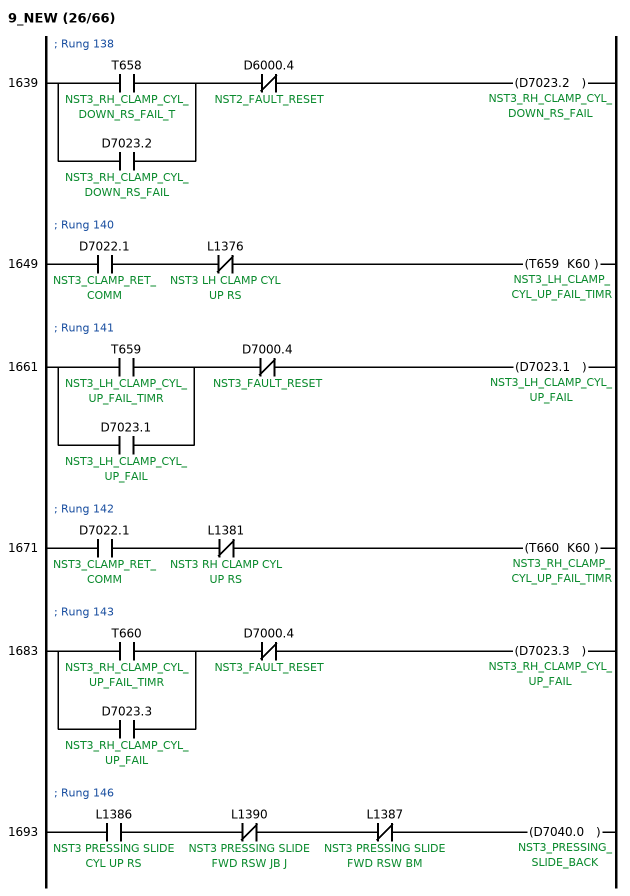
[picture p144: ladder of 9_NEW, rungs at steps 1639 to 1693]
; Rung 138
1639  LD      T658  ; NST3_RH_CLAMP_CYL_DOWN_RS_FAIL_T
      OR      D7023.2  ; NST3_RH_CLAMP_CYL_DOWN_RS_FAIL
      ANI     D6000.4  ; NST2_FAULT_RESET
      OUT     D7023.2  ; NST3_RH_CLAMP_CYL_DOWN_RS_FAIL
; Rung 140
1649  LD      D7022.1  ; NST3_CLAMP_RET_COMM
      ANI     L1376  ; NST3 LH CLAMP CYL UP RS
      OUT     T659 K60  ; NST3_LH_CLAMP_CYL_UP_FAIL_TIMR
; Rung 141
1661  LD      T659  ; NST3_LH_CLAMP_CYL_UP_FAIL_TIMR
      OR      D7023.1  ; NST3_LH_CLAMP_CYL_UP_FAIL
      ANI     D7000.4  ; NST3_FAULT_RESET
      OUT     D7023.1  ; NST3_LH_CLAMP_CYL_UP_FAIL
; Rung 142
1671  LD      D7022.1  ; NST3_CLAMP_RET_COMM
      ANI     L1381  ; NST3 RH CLAMP CYL UP RS
      OUT     T660 K60  ; NST3_RH_CLAMP_CYL_UP_FAIL_TIMR
; Rung 143
1683  LD      T660  ; NST3_RH_CLAMP_CYL_UP_FAIL_TIMR
      OR      D7023.3  ; NST3_RH_CLAMP_CYL_UP_FAIL
      ANI     D7000.4  ; NST3_FAULT_RESET
      OUT     D7023.3  ; NST3_RH_CLAMP_CYL_UP_FAIL
; Rung 146
1693  LD      L1386  ; NST3 PRESSING SLIDE CYL UP RS
      ANI     L1390  ; NST3 PRESSING SLIDE FWD RSW JB J
      ANI     L1387  ; NST3 PRESSING SLIDE FWD RSW BM
      OUT     D7040.0  ; NST3_PRESSING_SLIDE_BACK
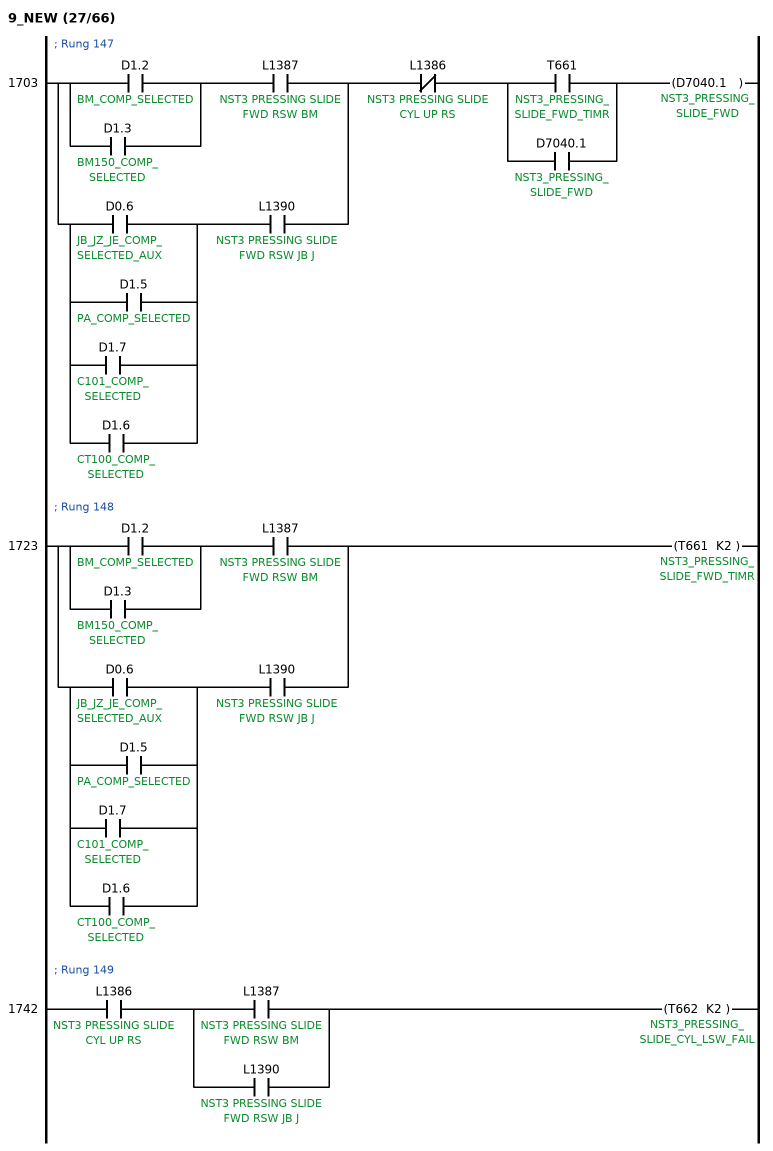
; Rung 147
1703  LD      D1.2  ; BM_COMP_SELECTED
      OR      D1.3  ; BM150_COMP_SELECTED
      AND     L1387  ; NST3 PRESSING SLIDE FWD RSW BM
      LD      D0.6  ; JB_JZ_JE_COMP_SELECTED_AUX
      OR      D1.5  ; PA_COMP_SELECTED
      OR      D1.7  ; C101_COMP_SELECTED
      OR      D1.6  ; CT100_COMP_SELECTED
      AND     L1390  ; NST3 PRESSING SLIDE FWD RSW JB J
      ORB
      ANI     L1386  ; NST3 PRESSING SLIDE CYL UP RS
      LD      T661  ; NST3_PRESSING_SLIDE_FWD_TIMR
      OR      D7040.1  ; NST3_PRESSING_SLIDE_FWD
      ANB
      OUT     D7040.1  ; NST3_PRESSING_SLIDE_FWD
; Rung 148
1723  LD      D1.2  ; BM_COMP_SELECTED
      OR      D1.3  ; BM150_COMP_SELECTED
      AND     L1387  ; NST3 PRESSING SLIDE FWD RSW BM
      LD      D0.6  ; JB_JZ_JE_COMP_SELECTED_AUX
      OR      D1.5  ; PA_COMP_SELECTED
      OR      D1.7  ; C101_COMP_SELECTED
      OR      D1.6  ; CT100_COMP_SELECTED
      AND     L1390  ; NST3 PRESSING SLIDE FWD RSW JB J
      ORB
      OUT     T661 K2  ; NST3_PRESSING_SLIDE_FWD_TIMR
; Rung 149
1742  LD      L1386  ; NST3 PRESSING SLIDE CYL UP RS
      LD      L1387  ; NST3 PRESSING SLIDE FWD RSW BM
      OR      L1390  ; NST3 PRESSING SLIDE FWD RSW JB J
      ANB
      OUT     T662 K2  ; NST3_PRESSING_SLIDE_CYL_LSW_FAIL
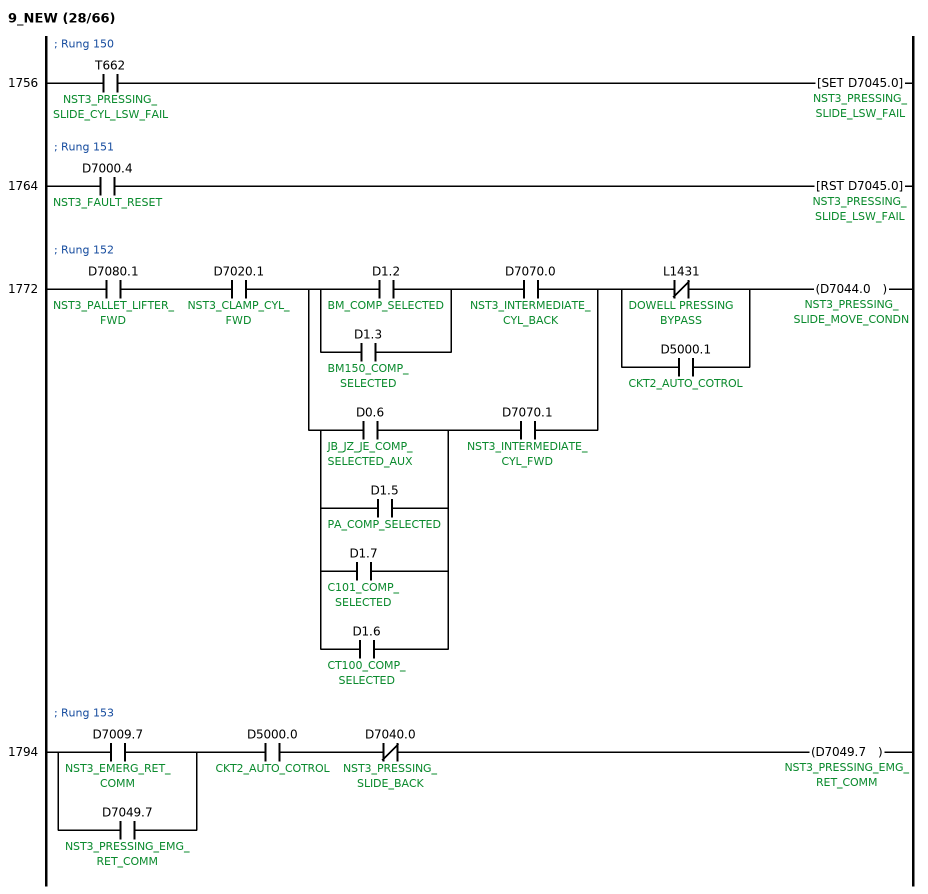
; Rung 150
1756  LD      T662  ; NST3_PRESSING_SLIDE_CYL_LSW_FAIL
      SET     D7045.0  ; NST3_PRESSING_SLIDE_LSW_FAIL
; Rung 151
1764  LD      D7000.4  ; NST3_FAULT_RESET
      RST     D7045.0  ; NST3_PRESSING_SLIDE_LSW_FAIL
; Rung 152
1772  LD      D7080.1  ; NST3_PALLET_LIFTER_FWD
      AND     D7020.1  ; NST3_CLAMP_CYL_FWD
      LD      D1.2  ; BM_COMP_SELECTED
      OR      D1.3  ; BM150_COMP_SELECTED
      AND     D7070.0  ; NST3_INTERMEDIATE_CYL_BACK
      LD      D0.6  ; JB_JZ_JE_COMP_SELECTED_AUX
      OR      D1.5  ; PA_COMP_SELECTED
      OR      D1.7  ; C101_COMP_SELECTED
      OR      D1.6  ; CT100_COMP_SELECTED
      AND     D7070.1  ; NST3_INTERMEDIATE_CYL_FWD
      ORB
      ANB
      LDI     L1431  ; DOWELL PRESSING BYPASS
      OR      D5000.1  ; CKT2_AUTO_COTROL
      ANB
      OUT     D7044.0  ; NST3_PRESSING_SLIDE_MOVE_CONDN
; Rung 153
1794  LD      D7009.7  ; NST3_EMERG_RET_COMM
      OR      D7049.7  ; NST3_PRESSING_EMG_RET_COMM
      AND     D5000.0  ; CKT2_AUTO_COTROL
      ANI     D7040.0  ; NST3_PRESSING_SLIDE_BACK
      OUT     D7049.7  ; NST3_PRESSING_EMG_RET_COMM
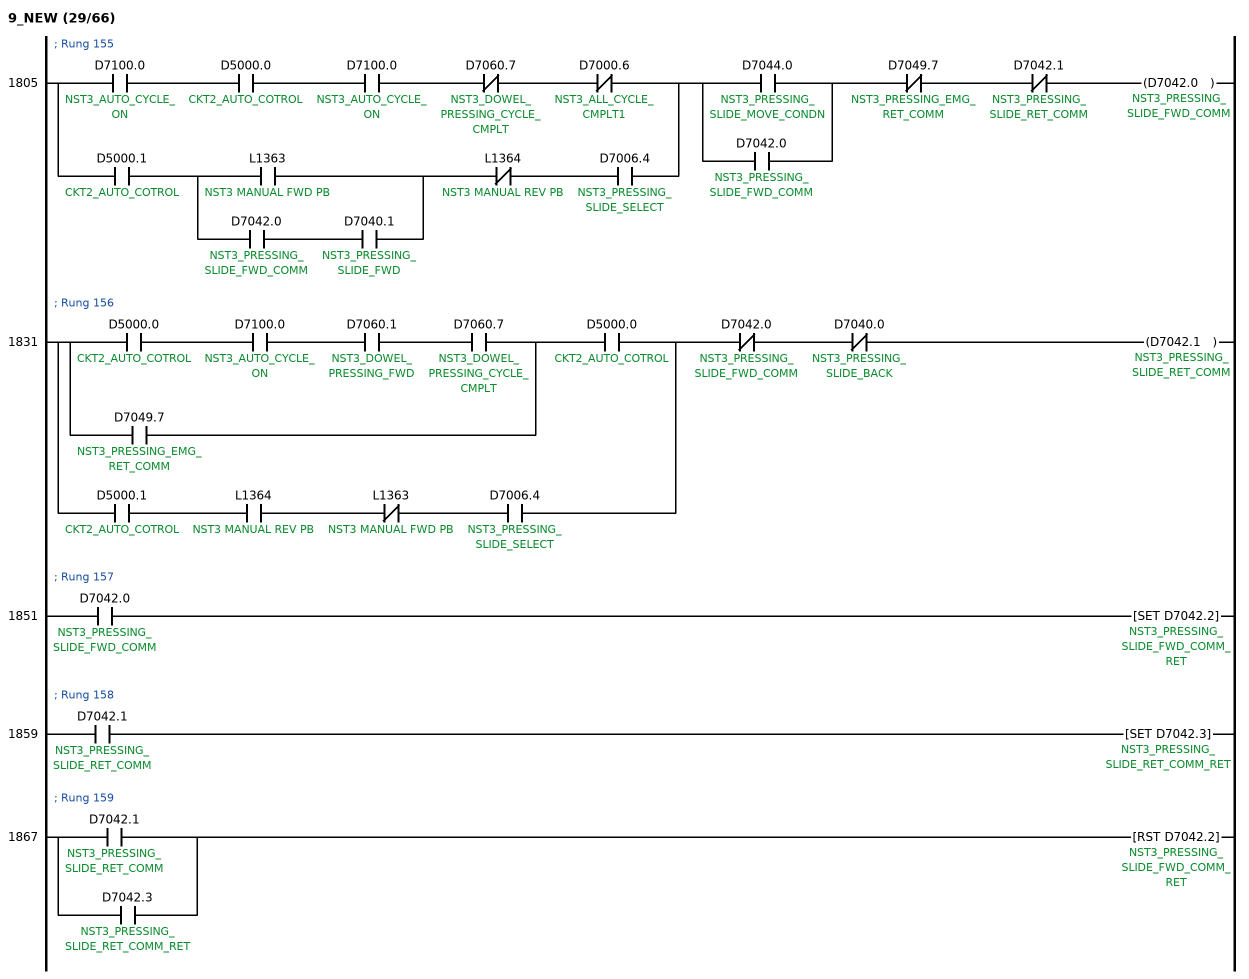
; Rung 155
1805  LD      D7100.0  ; NST3_AUTO_CYCLE_ON
      AND     D5000.0  ; CKT2_AUTO_COTROL
      AND     D7100.0  ; NST3_AUTO_CYCLE_ON
      ANI     D7060.7  ; NST3_DOWEL_PRESSING_CYCLE_CMPLT
      ANI     D7000.6  ; NST3_ALL_CYCLE_CMPLT1
      LD      D5000.1  ; CKT2_AUTO_COTROL
      LD      L1363  ; NST3 MANUAL FWD PB
      LD      D7042.0  ; NST3_PRESSING_SLIDE_FWD_COMM
      AND     D7040.1  ; NST3_PRESSING_SLIDE_FWD
      ORB
      ANB
      ANI     L1364  ; NST3 MANUAL REV PB
      AND     D7006.4  ; NST3_PRESSING_SLIDE_SELECT
      ORB
      LD      D7044.0  ; NST3_PRESSING_SLIDE_MOVE_CONDN
      OR      D7042.0  ; NST3_PRESSING_SLIDE_FWD_COMM
      ANB
      ANI     D7049.7  ; NST3_PRESSING_EMG_RET_COMM
      ANI     D7042.1  ; NST3_PRESSING_SLIDE_RET_COMM
      OUT     D7042.0  ; NST3_PRESSING_SLIDE_FWD_COMM
; Rung 156
1831  LD      D5000.0  ; CKT2_AUTO_COTROL
      AND     D7100.0  ; NST3_AUTO_CYCLE_ON
      AND     D7060.1  ; NST3_DOWEL_PRESSING_FWD
      AND     D7060.7  ; NST3_DOWEL_PRESSING_CYCLE_CMPLT
      OR      D7049.7  ; NST3_PRESSING_EMG_RET_COMM
      AND     D5000.0  ; CKT2_AUTO_COTROL
      LD      D5000.1  ; CKT2_AUTO_COTROL
      AND     L1364  ; NST3 MANUAL REV PB
      ANI     L1363  ; NST3 MANUAL FWD PB
      AND     D7006.4  ; NST3_PRESSING_SLIDE_SELECT
      ORB
      ANI     D7042.0  ; NST3_PRESSING_SLIDE_FWD_COMM
      ANI     D7040.0  ; NST3_PRESSING_SLIDE_BACK
      OUT     D7042.1  ; NST3_PRESSING_SLIDE_RET_COMM
; Rung 157
1851  LD      D7042.0  ; NST3_PRESSING_SLIDE_FWD_COMM
      SET     D7042.2  ; NST3_PRESSING_SLIDE_FWD_COMM_RET
; Rung 158
1859  LD      D7042.1  ; NST3_PRESSING_SLIDE_RET_COMM
      SET     D7042.3  ; NST3_PRESSING_SLIDE_RET_COMM_RET
; Rung 159
1867  LD      D7042.1  ; NST3_PRESSING_SLIDE_RET_COMM
      OR      D7042.3  ; NST3_PRESSING_SLIDE_RET_COMM_RET
      RST     D7042.2  ; NST3_PRESSING_SLIDE_FWD_COMM_RET
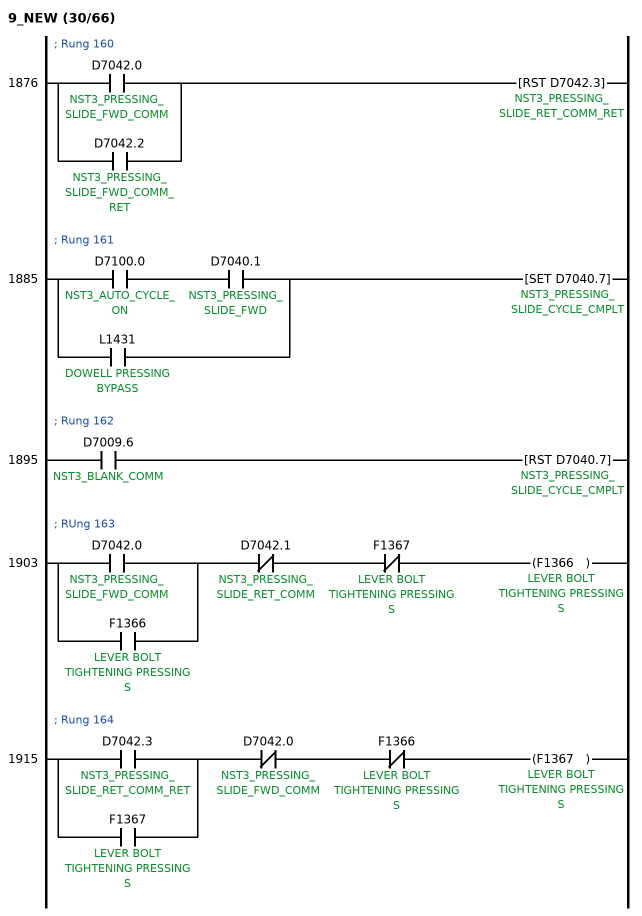
; Rung 160
1876  LD      D7042.0  ; NST3_PRESSING_SLIDE_FWD_COMM
      OR      D7042.2  ; NST3_PRESSING_SLIDE_FWD_COMM_RET
      RST     D7042.3  ; NST3_PRESSING_SLIDE_RET_COMM_RET
; Rung 161
1885  LD      D7100.0  ; NST3_AUTO_CYCLE_ON
      AND     D7040.1  ; NST3_PRESSING_SLIDE_FWD
      OR      L1431  ; DOWELL PRESSING BYPASS
      SET     D7040.7  ; NST3_PRESSING_SLIDE_CYCLE_CMPLT
; Rung 162
1895  LD      D7009.6  ; NST3_BLANK_COMM
      RST     D7040.7  ; NST3_PRESSING_SLIDE_CYCLE_CMPLT
; RUng 163
1903  LD      D7042.0  ; NST3_PRESSING_SLIDE_FWD_COMM
      OR      F1366  ; LEVER BOLT TIGHTENING PRESSING S
      ANI     D7042.1  ; NST3_PRESSING_SLIDE_RET_COMM
      ANI     F1367  ; LEVER BOLT TIGHTENING PRESSING S
      OUT     F1366  ; LEVER BOLT TIGHTENING PRESSING S
; Rung 164
1915  LD      D7042.3  ; NST3_PRESSING_SLIDE_RET_COMM_RET
      OR      F1367  ; LEVER BOLT TIGHTENING PRESSING S
      ANI     D7042.0  ; NST3_PRESSING_SLIDE_FWD_COMM
      ANI     F1366  ; LEVER BOLT TIGHTENING PRESSING S
      OUT     F1367  ; LEVER BOLT TIGHTENING PRESSING S
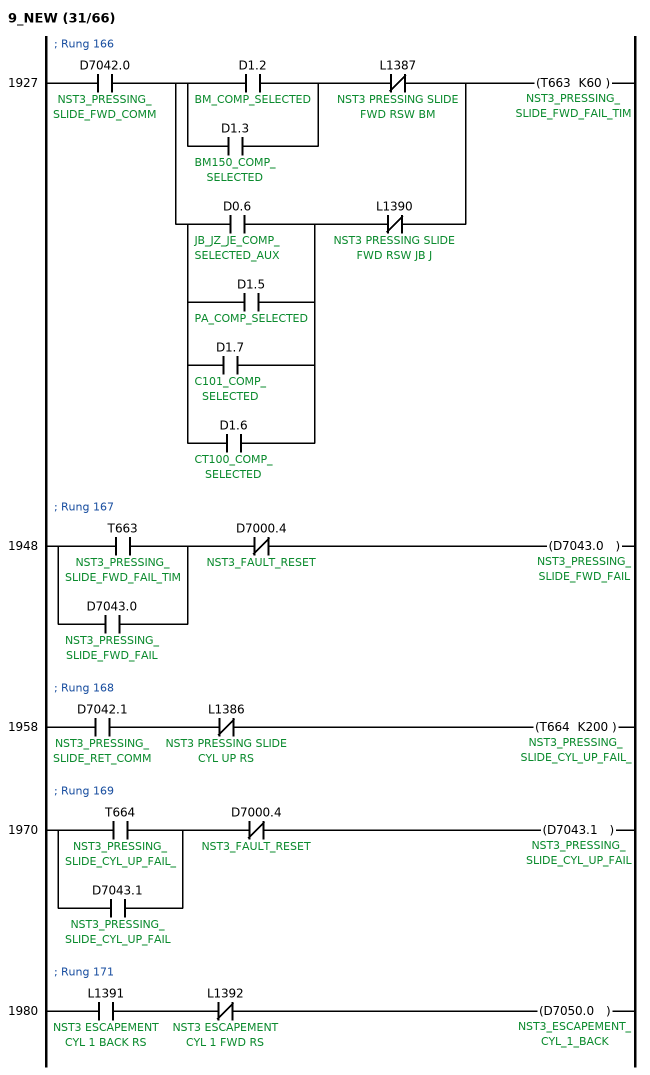
; Rung 166
1927  LD      D7042.0  ; NST3_PRESSING_SLIDE_FWD_COMM
      LD      D1.2  ; BM_COMP_SELECTED
      OR      D1.3  ; BM150_COMP_SELECTED
      ANI     L1387  ; NST3 PRESSING SLIDE FWD RSW BM
      LD      D0.6  ; JB_JZ_JE_COMP_SELECTED_AUX
      OR      D1.5  ; PA_COMP_SELECTED
      OR      D1.7  ; C101_COMP_SELECTED
      OR      D1.6  ; CT100_COMP_SELECTED
      ANI     L1390  ; NST3 PRESSING SLIDE FWD RSW JB J
      ORB
      ANB
      OUT     T663 K60  ; NST3_PRESSING_SLIDE_FWD_FAIL_TIM
; Rung 167
1948  LD      T663  ; NST3_PRESSING_SLIDE_FWD_FAIL_TIM
      OR      D7043.0  ; NST3_PRESSING_SLIDE_FWD_FAIL
      ANI     D7000.4  ; NST3_FAULT_RESET
      OUT     D7043.0  ; NST3_PRESSING_SLIDE_FWD_FAIL
; Rung 168
1958  LD      D7042.1  ; NST3_PRESSING_SLIDE_RET_COMM
      ANI     L1386  ; NST3 PRESSING SLIDE CYL UP RS
      OUT     T664 K200  ; NST3_PRESSING_SLIDE_CYL_UP_FAIL_
; Rung 169
1970  LD      T664  ; NST3_PRESSING_SLIDE_CYL_UP_FAIL_
      OR      D7043.1  ; NST3_PRESSING_SLIDE_CYL_UP_FAIL
      ANI     D7000.4  ; NST3_FAULT_RESET
      OUT     D7043.1  ; NST3_PRESSING_SLIDE_CYL_UP_FAIL
; Rung 171
1980  LD      L1391  ; NST3 ESCAPEMENT CYL 1 BACK RS
      ANI     L1392  ; NST3 ESCAPEMENT CYL 1 FWD RS
      OUT     D7050.0  ; NST3_ESCAPEMENT_CYL_1_BACK
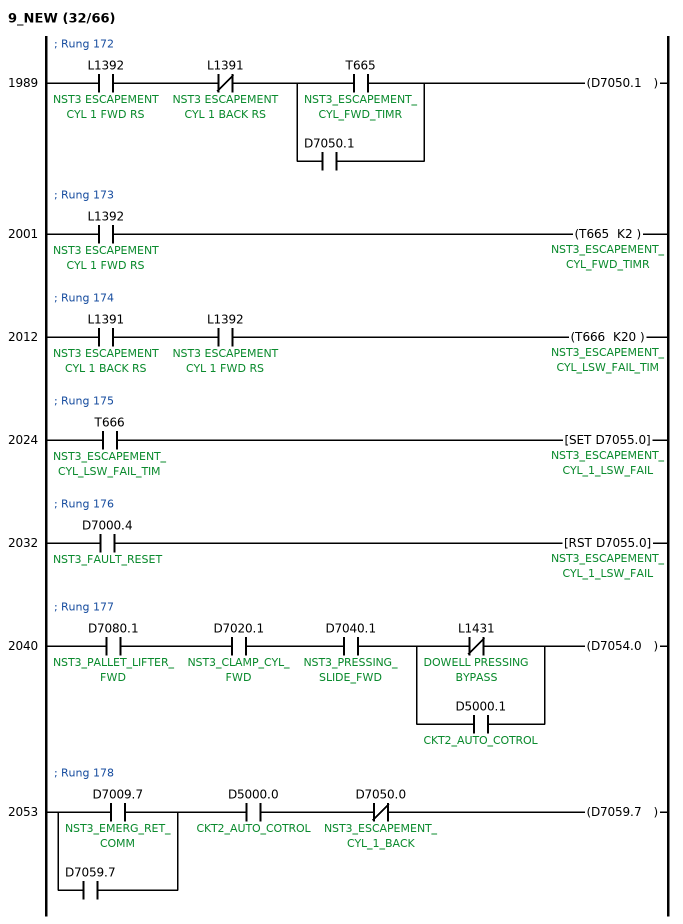
; Rung 172
1989  LD      L1392  ; NST3 ESCAPEMENT CYL 1 FWD RS
      ANI     L1391  ; NST3 ESCAPEMENT CYL 1 BACK RS
      LD      T665  ; NST3_ESCAPEMENT_CYL_FWD_TIMR
      OR      D7050.1
      ANB
      OUT     D7050.1
; Rung 173
2001  LD      L1392  ; NST3 ESCAPEMENT CYL 1 FWD RS
      OUT     T665 K2  ; NST3_ESCAPEMENT_CYL_FWD_TIMR
; Rung 174
2012  LD      L1391  ; NST3 ESCAPEMENT CYL 1 BACK RS
      AND     L1392  ; NST3 ESCAPEMENT CYL 1 FWD RS
      OUT     T666 K20  ; NST3_ESCAPEMENT_CYL_LSW_FAIL_TIM
; Rung 175
2024  LD      T666  ; NST3_ESCAPEMENT_CYL_LSW_FAIL_TIM
      SET     D7055.0  ; NST3_ESCAPEMENT_CYL_1_LSW_FAIL
; Rung 176
2032  LD      D7000.4  ; NST3_FAULT_RESET
      RST     D7055.0  ; NST3_ESCAPEMENT_CYL_1_LSW_FAIL
; Rung 177
2040  LD      D7080.1  ; NST3_PALLET_LIFTER_FWD
      AND     D7020.1  ; NST3_CLAMP_CYL_FWD
      AND     D7040.1  ; NST3_PRESSING_SLIDE_FWD
      LDI     L1431  ; DOWELL PRESSING BYPASS
      OR      D5000.1  ; CKT2_AUTO_COTROL
      ANB
      OUT     D7054.0
; Rung 178
2053  LD      D7009.7  ; NST3_EMERG_RET_COMM
      OR      D7059.7
      AND     D5000.0  ; CKT2_AUTO_COTROL
      ANI     D7050.0  ; NST3_ESCAPEMENT_CYL_1_BACK
      OUT     D7059.7
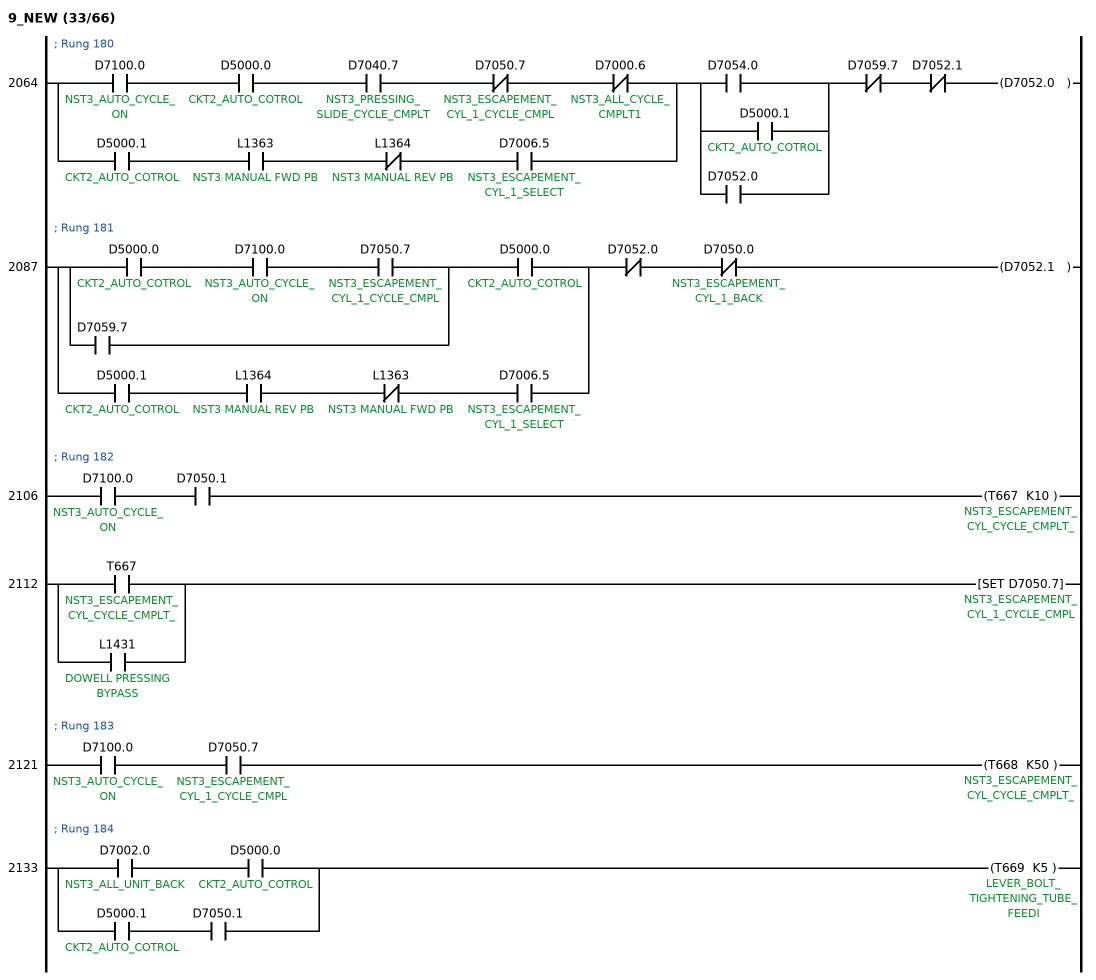
; Rung 180
2064  LD      D7100.0  ; NST3_AUTO_CYCLE_ON
      AND     D5000.0  ; CKT2_AUTO_COTROL
      AND     D7040.7  ; NST3_PRESSING_SLIDE_CYCLE_CMPLT
      ANI     D7050.7  ; NST3_ESCAPEMENT_CYL_1_CYCLE_CMPL
      ANI     D7000.6  ; NST3_ALL_CYCLE_CMPLT1
      LD      D5000.1  ; CKT2_AUTO_COTROL
      AND     L1363  ; NST3 MANUAL FWD PB
      ANI     L1364  ; NST3 MANUAL REV PB
      AND     D7006.5  ; NST3_ESCAPEMENT_CYL_1_SELECT
      ORB
      LD      D7054.0
      OR      D5000.1  ; CKT2_AUTO_COTROL
      OR      D7052.0
      ANB
      ANI     D7059.7
      ANI     D7052.1
      OUT     D7052.0
; Rung 181
2087  LD      D5000.0  ; CKT2_AUTO_COTROL
      AND     D7100.0  ; NST3_AUTO_CYCLE_ON
      AND     D7050.7  ; NST3_ESCAPEMENT_CYL_1_CYCLE_CMPL
      OR      D7059.7
      AND     D5000.0  ; CKT2_AUTO_COTROL
      LD      D5000.1  ; CKT2_AUTO_COTROL
      AND     L1364  ; NST3 MANUAL REV PB
      ANI     L1363  ; NST3 MANUAL FWD PB
      AND     D7006.5  ; NST3_ESCAPEMENT_CYL_1_SELECT
      ORB
      ANI     D7052.0
      ANI     D7050.0  ; NST3_ESCAPEMENT_CYL_1_BACK
      OUT     D7052.1
; Rung 182
2106  LD      D7100.0  ; NST3_AUTO_CYCLE_ON
      AND     D7050.1
      OUT     T667 K10  ; NST3_ESCAPEMENT_CYL_CYCLE_CMPLT_
2112  LD      T667  ; NST3_ESCAPEMENT_CYL_CYCLE_CMPLT_
      OR      L1431  ; DOWELL PRESSING BYPASS
      SET     D7050.7  ; NST3_ESCAPEMENT_CYL_1_CYCLE_CMPL
; Rung 183
2121  LD      D7100.0  ; NST3_AUTO_CYCLE_ON
      AND     D7050.7  ; NST3_ESCAPEMENT_CYL_1_CYCLE_CMPL
      OUT     T668 K50  ; NST3_ESCAPEMENT_CYL_CYCLE_CMPLT_
; Rung 184
2133  LD      D7002.0  ; NST3_ALL_UNIT_BACK
      AND     D5000.0  ; CKT2_AUTO_COTROL
      LD      D5000.1  ; CKT2_AUTO_COTROL
      AND     D7050.1
      ORB
      OUT     T669 K5  ; LEVER_BOLT_TIGHTENING_TUBE_FEEDI
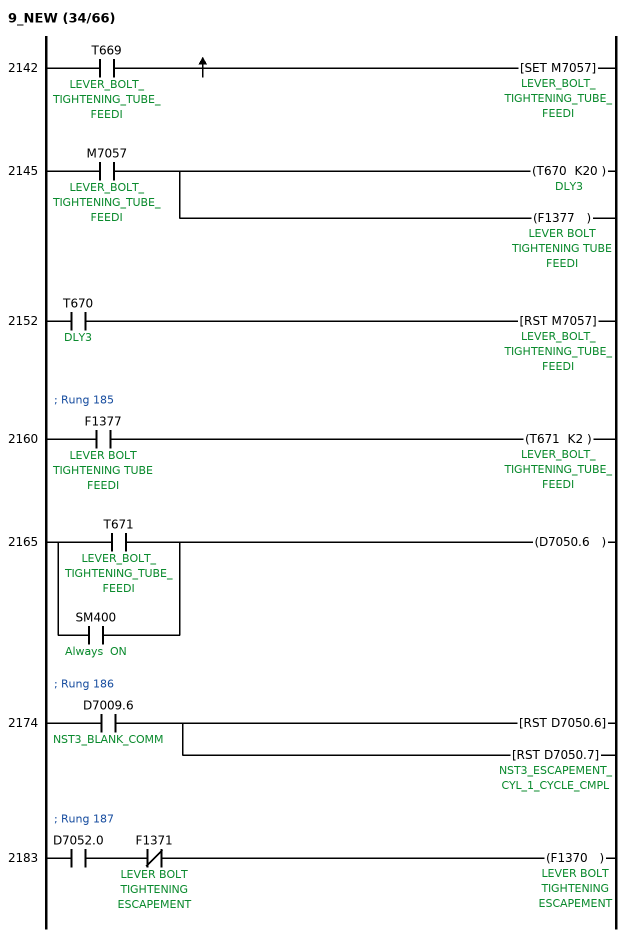
2142  LD      T669  ; LEVER_BOLT_TIGHTENING_TUBE_FEEDI
      MEP
      SET     M7057  ; LEVER_BOLT_TIGHTENING_TUBE_FEEDI
2145  LD      M7057  ; LEVER_BOLT_TIGHTENING_TUBE_FEEDI
      OUT     T670 K20  ; DLY3
      OUT     F1377  ; LEVER BOLT TIGHTENING TUBE FEEDI
2152  LD      T670  ; DLY3
      RST     M7057  ; LEVER_BOLT_TIGHTENING_TUBE_FEEDI
; Rung 185
2160  LD      F1377  ; LEVER BOLT TIGHTENING TUBE FEEDI
      OUT     T671 K2  ; LEVER_BOLT_TIGHTENING_TUBE_FEEDI
2165  LD      T671  ; LEVER_BOLT_TIGHTENING_TUBE_FEEDI
      OR      SM400  ; Always  ON
      OUT     D7050.6
; Rung 186
2174  LD      D7009.6  ; NST3_BLANK_COMM
      RST     D7050.6
      RST     D7050.7  ; NST3_ESCAPEMENT_CYL_1_CYCLE_CMPL
; Rung 187
2183  LD      D7052.0
      ANI     F1371  ; LEVER BOLT TIGHTENING ESCAPEMENT
      OUT     F1370  ; LEVER BOLT TIGHTENING ESCAPEMENT
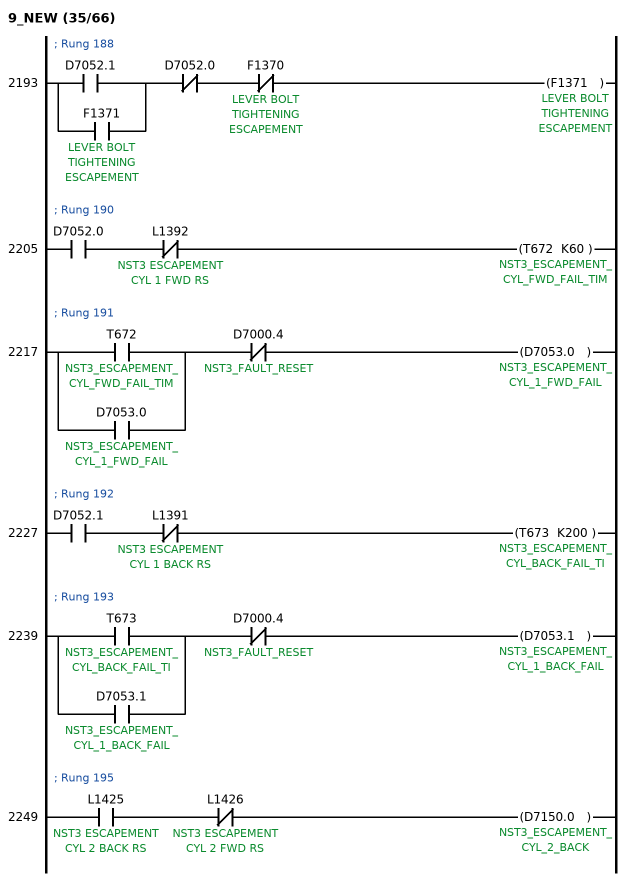
; Rung 188
2193  LD      D7052.1
      OR      F1371  ; LEVER BOLT TIGHTENING ESCAPEMENT
      ANI     D7052.0
      ANI     F1370  ; LEVER BOLT TIGHTENING ESCAPEMENT
      OUT     F1371  ; LEVER BOLT TIGHTENING ESCAPEMENT
; Rung 190
2205  LD      D7052.0
      ANI     L1392  ; NST3 ESCAPEMENT CYL 1 FWD RS
      OUT     T672 K60  ; NST3_ESCAPEMENT_CYL_FWD_FAIL_TIM
; Rung 191
2217  LD      T672  ; NST3_ESCAPEMENT_CYL_FWD_FAIL_TIM
      OR      D7053.0  ; NST3_ESCAPEMENT_CYL_1_FWD_FAIL
      ANI     D7000.4  ; NST3_FAULT_RESET
      OUT     D7053.0  ; NST3_ESCAPEMENT_CYL_1_FWD_FAIL
; Rung 192
2227  LD      D7052.1
      ANI     L1391  ; NST3 ESCAPEMENT CYL 1 BACK RS
      OUT     T673 K200  ; NST3_ESCAPEMENT_CYL_BACK_FAIL_TI
; Rung 193
2239  LD      T673  ; NST3_ESCAPEMENT_CYL_BACK_FAIL_TI
      OR      D7053.1  ; NST3_ESCAPEMENT_CYL_1_BACK_FAIL
      ANI     D7000.4  ; NST3_FAULT_RESET
      OUT     D7053.1  ; NST3_ESCAPEMENT_CYL_1_BACK_FAIL
; Rung 195
2249  LD      L1425  ; NST3 ESCAPEMENT CYL 2 BACK RS
      ANI     L1426  ; NST3 ESCAPEMENT CYL 2 FWD RS
      OUT     D7150.0  ; NST3_ESCAPEMENT_CYL_2_BACK
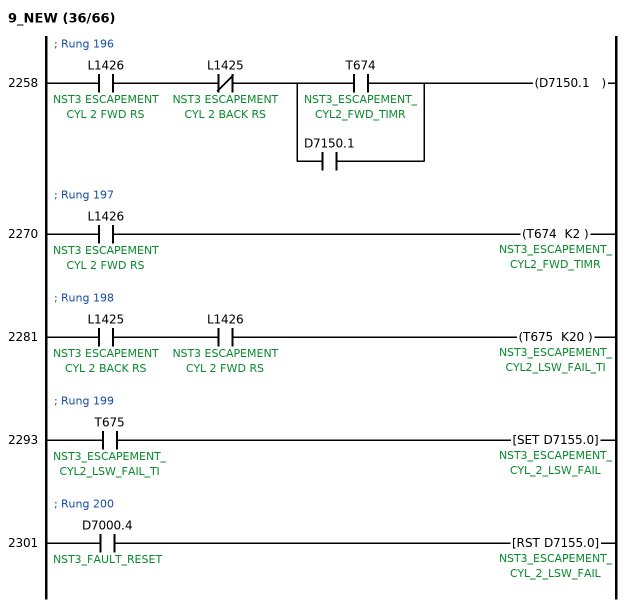
; Rung 196
2258  LD      L1426  ; NST3 ESCAPEMENT CYL 2 FWD RS
      ANI     L1425  ; NST3 ESCAPEMENT CYL 2 BACK RS
      LD      T674  ; NST3_ESCAPEMENT_CYL2_FWD_TIMR
      OR      D7150.1
      ANB
      OUT     D7150.1
; Rung 197
2270  LD      L1426  ; NST3 ESCAPEMENT CYL 2 FWD RS
      OUT     T674 K2  ; NST3_ESCAPEMENT_CYL2_FWD_TIMR
; Rung 198
2281  LD      L1425  ; NST3 ESCAPEMENT CYL 2 BACK RS
      AND     L1426  ; NST3 ESCAPEMENT CYL 2 FWD RS
      OUT     T675 K20  ; NST3_ESCAPEMENT_CYL2_LSW_FAIL_TI
; Rung 199
2293  LD      T675  ; NST3_ESCAPEMENT_CYL2_LSW_FAIL_TI
      SET     D7155.0  ; NST3_ESCAPEMENT_CYL_2_LSW_FAIL
; Rung 200
2301  LD      D7000.4  ; NST3_FAULT_RESET
      RST     D7155.0  ; NST3_ESCAPEMENT_CYL_2_LSW_FAIL
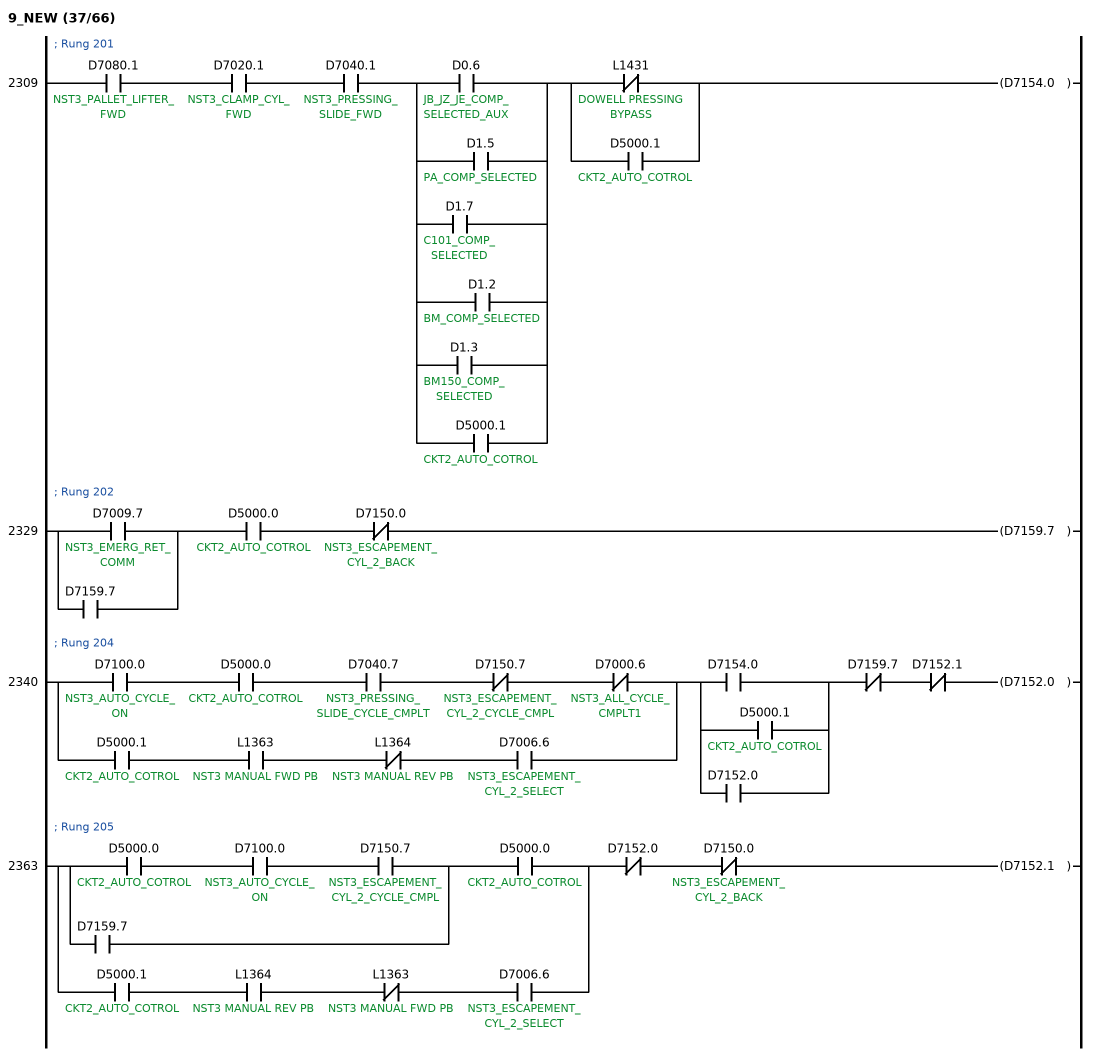
; Rung 201
2309  LD      D7080.1  ; NST3_PALLET_LIFTER_FWD
      AND     D7020.1  ; NST3_CLAMP_CYL_FWD
      AND     D7040.1  ; NST3_PRESSING_SLIDE_FWD
      LD      D0.6  ; JB_JZ_JE_COMP_SELECTED_AUX
      OR      D1.5  ; PA_COMP_SELECTED
      OR      D1.7  ; C101_COMP_SELECTED
      OR      D1.2  ; BM_COMP_SELECTED
      OR      D1.3  ; BM150_COMP_SELECTED
      OR      D5000.1  ; CKT2_AUTO_COTROL
      ANB
      LDI     L1431  ; DOWELL PRESSING BYPASS
      OR      D5000.1  ; CKT2_AUTO_COTROL
      ANB
      OUT     D7154.0
; Rung 202
2329  LD      D7009.7  ; NST3_EMERG_RET_COMM
      OR      D7159.7
      AND     D5000.0  ; CKT2_AUTO_COTROL
      ANI     D7150.0  ; NST3_ESCAPEMENT_CYL_2_BACK
      OUT     D7159.7
; Rung 204
2340  LD      D7100.0  ; NST3_AUTO_CYCLE_ON
      AND     D5000.0  ; CKT2_AUTO_COTROL
      AND     D7040.7  ; NST3_PRESSING_SLIDE_CYCLE_CMPLT
      ANI     D7150.7  ; NST3_ESCAPEMENT_CYL_2_CYCLE_CMPL
      ANI     D7000.6  ; NST3_ALL_CYCLE_CMPLT1
      LD      D5000.1  ; CKT2_AUTO_COTROL
      AND     L1363  ; NST3 MANUAL FWD PB
      ANI     L1364  ; NST3 MANUAL REV PB
      AND     D7006.6  ; NST3_ESCAPEMENT_CYL_2_SELECT
      ORB
      LD      D7154.0
      OR      D5000.1  ; CKT2_AUTO_COTROL
      OR      D7152.0
      ANB
      ANI     D7159.7
      ANI     D7152.1
      OUT     D7152.0
; Rung 205
2363  LD      D5000.0  ; CKT2_AUTO_COTROL
      AND     D7100.0  ; NST3_AUTO_CYCLE_ON
      AND     D7150.7  ; NST3_ESCAPEMENT_CYL_2_CYCLE_CMPL
      OR      D7159.7
      AND     D5000.0  ; CKT2_AUTO_COTROL
      LD      D5000.1  ; CKT2_AUTO_COTROL
      AND     L1364  ; NST3 MANUAL REV PB
      ANI     L1363  ; NST3 MANUAL FWD PB
      AND     D7006.6  ; NST3_ESCAPEMENT_CYL_2_SELECT
      ORB
      ANI     D7152.0
      ANI     D7150.0  ; NST3_ESCAPEMENT_CYL_2_BACK
      OUT     D7152.1
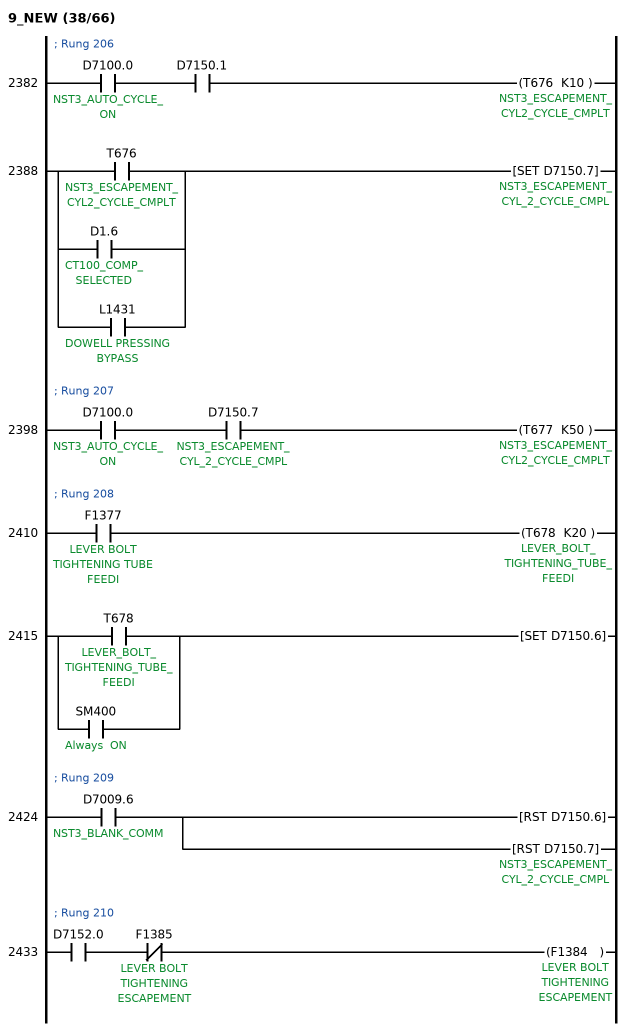
; Rung 206
2382  LD      D7100.0  ; NST3_AUTO_CYCLE_ON
      AND     D7150.1
      OUT     T676 K10  ; NST3_ESCAPEMENT_CYL2_CYCLE_CMPLT
2388  LD      T676  ; NST3_ESCAPEMENT_CYL2_CYCLE_CMPLT
      OR      D1.6  ; CT100_COMP_SELECTED
      OR      L1431  ; DOWELL PRESSING BYPASS
      SET     D7150.7  ; NST3_ESCAPEMENT_CYL_2_CYCLE_CMPL
; Rung 207
2398  LD      D7100.0  ; NST3_AUTO_CYCLE_ON
      AND     D7150.7  ; NST3_ESCAPEMENT_CYL_2_CYCLE_CMPL
      OUT     T677 K50  ; NST3_ESCAPEMENT_CYL2_CYCLE_CMPLT
; Rung 208
2410  LD      F1377  ; LEVER BOLT TIGHTENING TUBE FEEDI
      OUT     T678 K20  ; LEVER_BOLT_TIGHTENING_TUBE_FEEDI
2415  LD      T678  ; LEVER_BOLT_TIGHTENING_TUBE_FEEDI
      OR      SM400  ; Always  ON
      SET     D7150.6
; Rung 209
2424  LD      D7009.6  ; NST3_BLANK_COMM
      RST     D7150.6
      RST     D7150.7  ; NST3_ESCAPEMENT_CYL_2_CYCLE_CMPL
; Rung 210
2433  LD      D7152.0
      ANI     F1385  ; LEVER BOLT TIGHTENING ESCAPEMENT
      OUT     F1384  ; LEVER BOLT TIGHTENING ESCAPEMENT
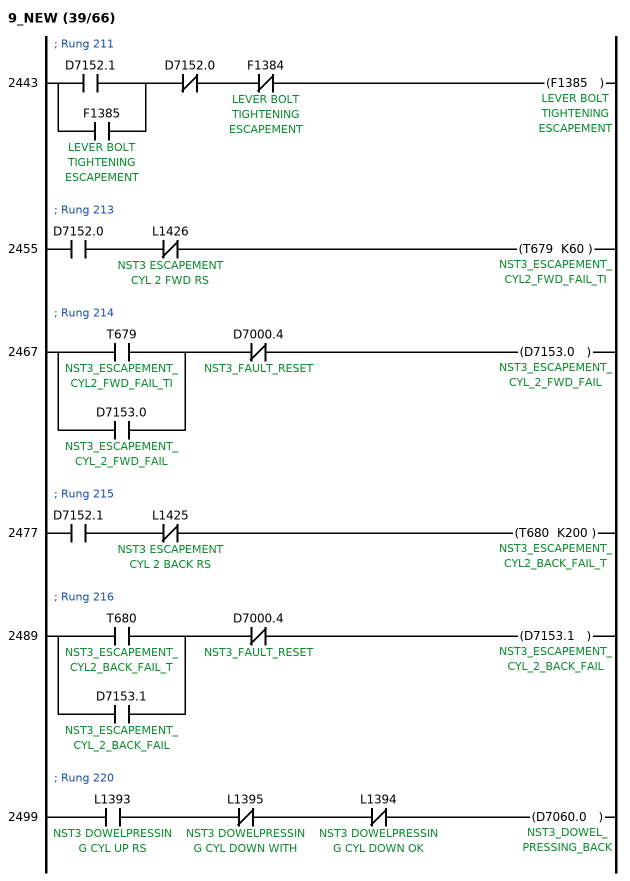
; Rung 211
2443  LD      D7152.1
      OR      F1385  ; LEVER BOLT TIGHTENING ESCAPEMENT
      ANI     D7152.0
      ANI     F1384  ; LEVER BOLT TIGHTENING ESCAPEMENT
      OUT     F1385  ; LEVER BOLT TIGHTENING ESCAPEMENT
; Rung 213
2455  LD      D7152.0
      ANI     L1426  ; NST3 ESCAPEMENT CYL 2 FWD RS
      OUT     T679 K60  ; NST3_ESCAPEMENT_CYL2_FWD_FAIL_TI
; Rung 214
2467  LD      T679  ; NST3_ESCAPEMENT_CYL2_FWD_FAIL_TI
      OR      D7153.0  ; NST3_ESCAPEMENT_CYL_2_FWD_FAIL
      ANI     D7000.4  ; NST3_FAULT_RESET
      OUT     D7153.0  ; NST3_ESCAPEMENT_CYL_2_FWD_FAIL
; Rung 215
2477  LD      D7152.1
      ANI     L1425  ; NST3 ESCAPEMENT CYL 2 BACK RS
      OUT     T680 K200  ; NST3_ESCAPEMENT_CYL2_BACK_FAIL_T
; Rung 216
2489  LD      T680  ; NST3_ESCAPEMENT_CYL2_BACK_FAIL_T
      OR      D7153.1  ; NST3_ESCAPEMENT_CYL_2_BACK_FAIL
      ANI     D7000.4  ; NST3_FAULT_RESET
      OUT     D7153.1  ; NST3_ESCAPEMENT_CYL_2_BACK_FAIL
; Rung 220
2499  LD      L1393  ; NST3 DOWELPRESSING CYL UP RS
      ANI     L1395  ; NST3 DOWELPRESSING CYL DOWN WITH
      ANI     L1394  ; NST3 DOWELPRESSING CYL DOWN OK
      OUT     D7060.0  ; NST3_DOWEL_PRESSING_BACK
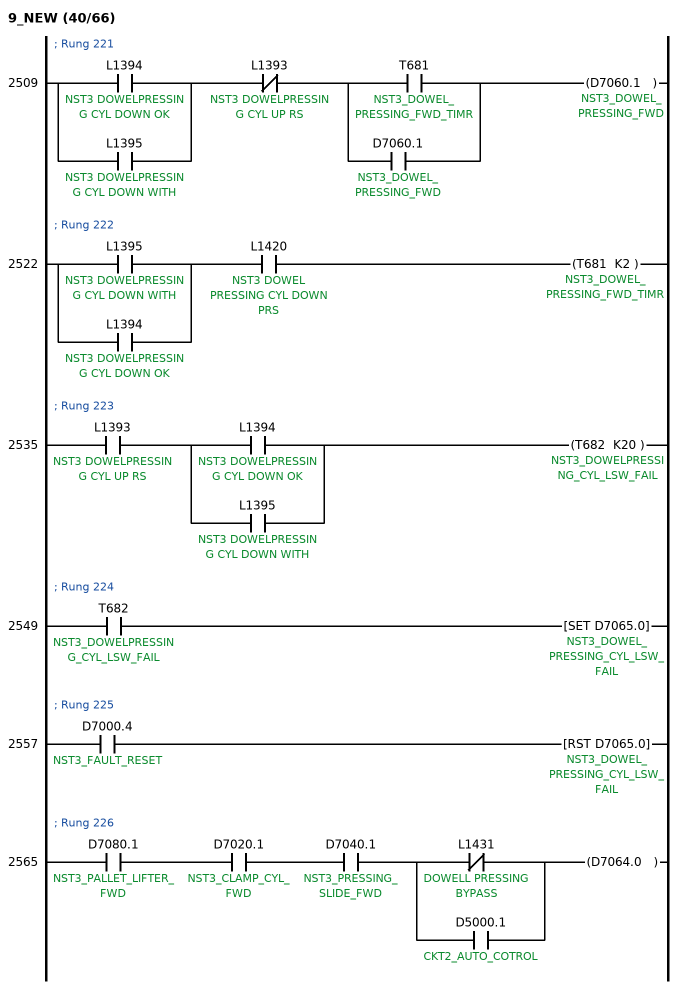
; Rung 221
2509  LD      L1394  ; NST3 DOWELPRESSING CYL DOWN OK
      OR      L1395  ; NST3 DOWELPRESSING CYL DOWN WITH
      ANI     L1393  ; NST3 DOWELPRESSING CYL UP RS
      LD      T681  ; NST3_DOWEL_PRESSING_FWD_TIMR
      OR      D7060.1  ; NST3_DOWEL_PRESSING_FWD
      ANB
      OUT     D7060.1  ; NST3_DOWEL_PRESSING_FWD
; Rung 222
2522  LD      L1395  ; NST3 DOWELPRESSING CYL DOWN WITH
      OR      L1394  ; NST3 DOWELPRESSING CYL DOWN OK
      AND     L1420  ; NST3 DOWEL PRESSING CYL DOWN PRS
      OUT     T681 K2  ; NST3_DOWEL_PRESSING_FWD_TIMR
; Rung 223
2535  LD      L1393  ; NST3 DOWELPRESSING CYL UP RS
      LD      L1394  ; NST3 DOWELPRESSING CYL DOWN OK
      OR      L1395  ; NST3 DOWELPRESSING CYL DOWN WITH
      ANB
      OUT     T682 K20  ; NST3_DOWELPRESSING_CYL_LSW_FAIL
; Rung 224
2549  LD      T682  ; NST3_DOWELPRESSING_CYL_LSW_FAIL
      SET     D7065.0  ; NST3_DOWEL_PRESSING_CYL_LSW_FAIL
; Rung 225
2557  LD      D7000.4  ; NST3_FAULT_RESET
      RST     D7065.0  ; NST3_DOWEL_PRESSING_CYL_LSW_FAIL
; Rung 226
2565  LD      D7080.1  ; NST3_PALLET_LIFTER_FWD
      AND     D7020.1  ; NST3_CLAMP_CYL_FWD
      AND     D7040.1  ; NST3_PRESSING_SLIDE_FWD
      LDI     L1431  ; DOWELL PRESSING BYPASS
      OR      D5000.1  ; CKT2_AUTO_COTROL
      ANB
      OUT     D7064.0
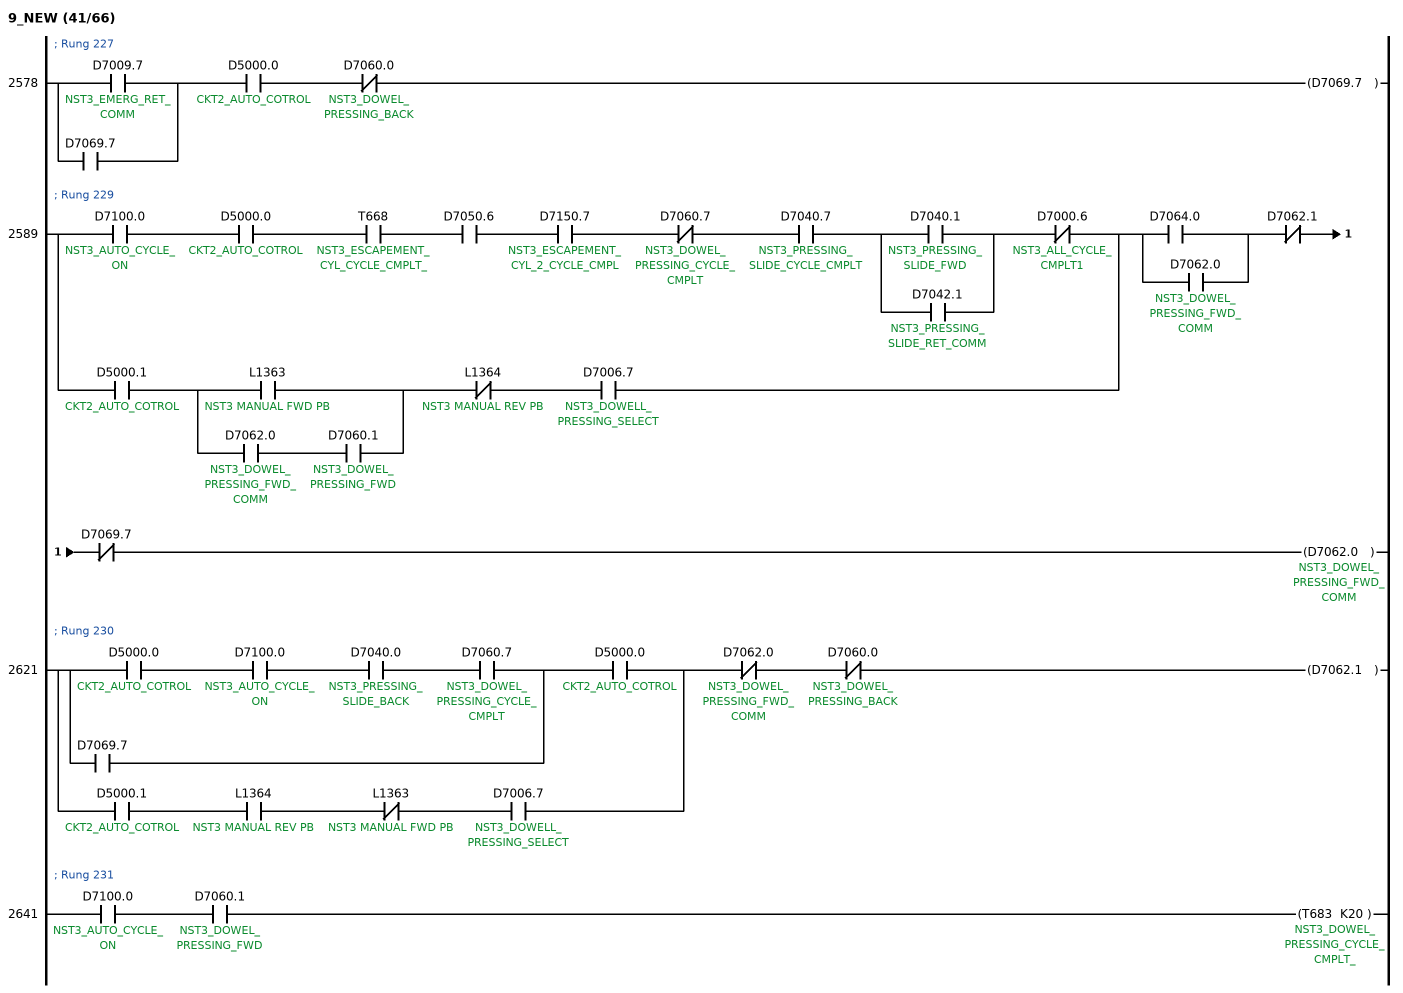
; Rung 227
2578  LD      D7009.7  ; NST3_EMERG_RET_COMM
      OR      D7069.7
      AND     D5000.0  ; CKT2_AUTO_COTROL
      ANI     D7060.0  ; NST3_DOWEL_PRESSING_BACK
      OUT     D7069.7
; Rung 229
2589  LD      D7100.0  ; NST3_AUTO_CYCLE_ON
      AND     D5000.0  ; CKT2_AUTO_COTROL
      AND     T668  ; NST3_ESCAPEMENT_CYL_CYCLE_CMPLT_
      AND     D7050.6
      AND     D7150.7  ; NST3_ESCAPEMENT_CYL_2_CYCLE_CMPL
      ANI     D7060.7  ; NST3_DOWEL_PRESSING_CYCLE_CMPLT
      AND     D7040.7  ; NST3_PRESSING_SLIDE_CYCLE_CMPLT
      LD      D7040.1  ; NST3_PRESSING_SLIDE_FWD
      OR      D7042.1  ; NST3_PRESSING_SLIDE_RET_COMM
      ANB
      ANI     D7000.6  ; NST3_ALL_CYCLE_CMPLT1
      LD      D5000.1  ; CKT2_AUTO_COTROL
      LD      L1363  ; NST3 MANUAL FWD PB
      LD      D7062.0  ; NST3_DOWEL_PRESSING_FWD_COMM
      AND     D7060.1  ; NST3_DOWEL_PRESSING_FWD
      ORB
      ANB
      ANI     L1364  ; NST3 MANUAL REV PB
      AND     D7006.7  ; NST3_DOWELL_PRESSING_SELECT
      ORB
      LD      D7064.0
      OR      D7062.0  ; NST3_DOWEL_PRESSING_FWD_COMM
      ANB
      ANI     D7062.1
      ANI     D7069.7
      OUT     D7062.0  ; NST3_DOWEL_PRESSING_FWD_COMM
; Rung 230
2621  LD      D5000.0  ; CKT2_AUTO_COTROL
      AND     D7100.0  ; NST3_AUTO_CYCLE_ON
      AND     D7040.0  ; NST3_PRESSING_SLIDE_BACK
      AND     D7060.7  ; NST3_DOWEL_PRESSING_CYCLE_CMPLT
      OR      D7069.7
      AND     D5000.0  ; CKT2_AUTO_COTROL
      LD      D5000.1  ; CKT2_AUTO_COTROL
      AND     L1364  ; NST3 MANUAL REV PB
      ANI     L1363  ; NST3 MANUAL FWD PB
      AND     D7006.7  ; NST3_DOWELL_PRESSING_SELECT
      ORB
      ANI     D7062.0  ; NST3_DOWEL_PRESSING_FWD_COMM
      ANI     D7060.0  ; NST3_DOWEL_PRESSING_BACK
      OUT     D7062.1
; Rung 231
2641  LD      D7100.0  ; NST3_AUTO_CYCLE_ON
      AND     D7060.1  ; NST3_DOWEL_PRESSING_FWD
      OUT     T683 K20  ; NST3_DOWEL_PRESSING_CYCLE_CMPLT_
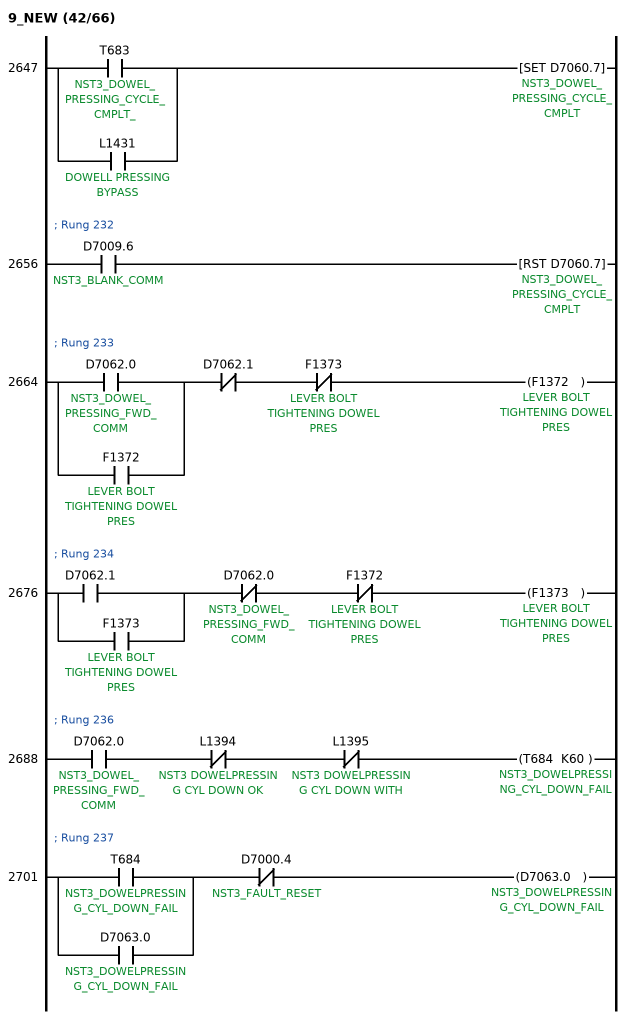
2647  LD      T683  ; NST3_DOWEL_PRESSING_CYCLE_CMPLT_
      OR      L1431  ; DOWELL PRESSING BYPASS
      SET     D7060.7  ; NST3_DOWEL_PRESSING_CYCLE_CMPLT
; Rung 232
2656  LD      D7009.6  ; NST3_BLANK_COMM
      RST     D7060.7  ; NST3_DOWEL_PRESSING_CYCLE_CMPLT
; Rung 233
2664  LD      D7062.0  ; NST3_DOWEL_PRESSING_FWD_COMM
      OR      F1372  ; LEVER BOLT TIGHTENING DOWEL PRES
      ANI     D7062.1
      ANI     F1373  ; LEVER BOLT TIGHTENING DOWEL PRES
      OUT     F1372  ; LEVER BOLT TIGHTENING DOWEL PRES
; Rung 234
2676  LD      D7062.1
      OR      F1373  ; LEVER BOLT TIGHTENING DOWEL PRES
      ANI     D7062.0  ; NST3_DOWEL_PRESSING_FWD_COMM
      ANI     F1372  ; LEVER BOLT TIGHTENING DOWEL PRES
      OUT     F1373  ; LEVER BOLT TIGHTENING DOWEL PRES
; Rung 236
2688  LD      D7062.0  ; NST3_DOWEL_PRESSING_FWD_COMM
      ANI     L1394  ; NST3 DOWELPRESSING CYL DOWN OK
      ANI     L1395  ; NST3 DOWELPRESSING CYL DOWN WITH
      OUT     T684 K60  ; NST3_DOWELPRESSING_CYL_DOWN_FAIL
; Rung 237
2701  LD      T684  ; NST3_DOWELPRESSING_CYL_DOWN_FAIL
      OR      D7063.0  ; NST3_DOWELPRESSING_CYL_DOWN_FAIL
      ANI     D7000.4  ; NST3_FAULT_RESET
      OUT     D7063.0  ; NST3_DOWELPRESSING_CYL_DOWN_FAIL
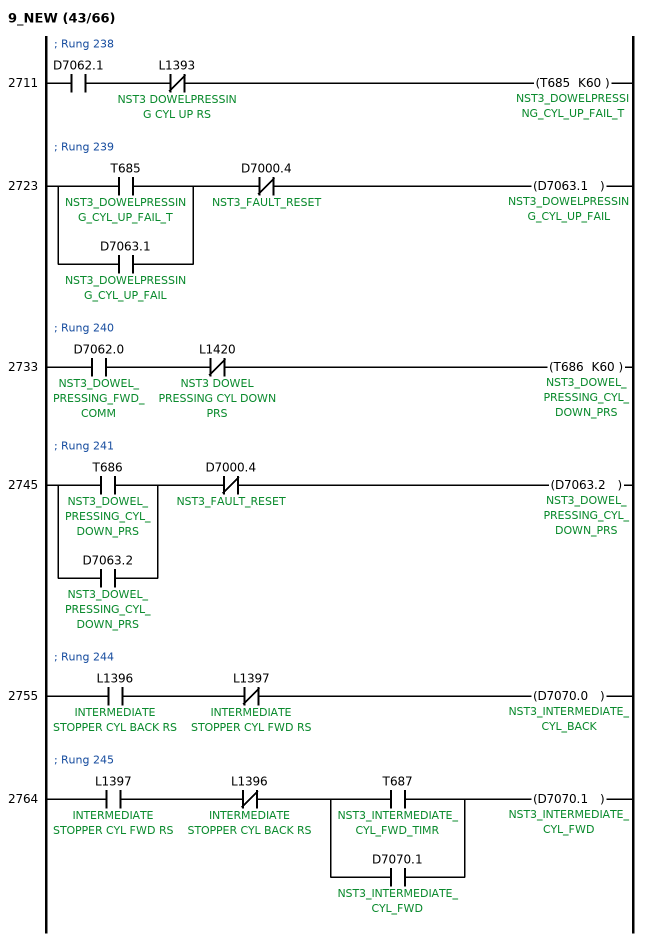
; Rung 238
2711  LD      D7062.1
      ANI     L1393  ; NST3 DOWELPRESSING CYL UP RS
      OUT     T685 K60  ; NST3_DOWELPRESSING_CYL_UP_FAIL_T
; Rung 239
2723  LD      T685  ; NST3_DOWELPRESSING_CYL_UP_FAIL_T
      OR      D7063.1  ; NST3_DOWELPRESSING_CYL_UP_FAIL
      ANI     D7000.4  ; NST3_FAULT_RESET
      OUT     D7063.1  ; NST3_DOWELPRESSING_CYL_UP_FAIL
; Rung 240
2733  LD      D7062.0  ; NST3_DOWEL_PRESSING_FWD_COMM
      ANI     L1420  ; NST3 DOWEL PRESSING CYL DOWN PRS
      OUT     T686 K60  ; NST3_DOWEL_PRESSING_CYL_DOWN_PRS
; Rung 241
2745  LD      T686  ; NST3_DOWEL_PRESSING_CYL_DOWN_PRS
      OR      D7063.2  ; NST3_DOWEL_PRESSING_CYL_DOWN_PRS
      ANI     D7000.4  ; NST3_FAULT_RESET
      OUT     D7063.2  ; NST3_DOWEL_PRESSING_CYL_DOWN_PRS
; Rung 244
2755  LD      L1396  ; INTERMEDIATE STOPPER CYL BACK RS
      ANI     L1397  ; INTERMEDIATE STOPPER CYL FWD RS
      OUT     D7070.0  ; NST3_INTERMEDIATE_CYL_BACK
; Rung 245
2764  LD      L1397  ; INTERMEDIATE STOPPER CYL FWD RS
      ANI     L1396  ; INTERMEDIATE STOPPER CYL BACK RS
      LD      T687  ; NST3_INTERMEDIATE_CYL_FWD_TIMR
      OR      D7070.1  ; NST3_INTERMEDIATE_CYL_FWD
      ANB
      OUT     D7070.1  ; NST3_INTERMEDIATE_CYL_FWD
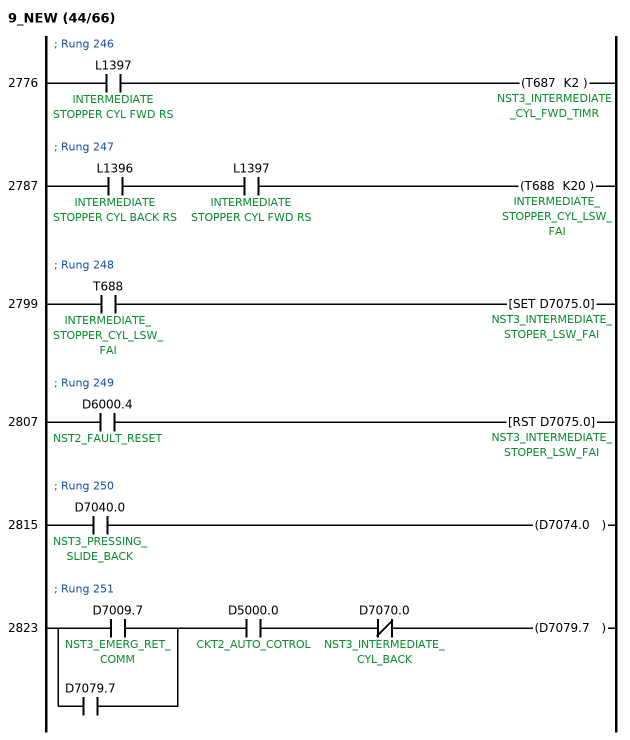
; Rung 246
2776  LD      L1397  ; INTERMEDIATE STOPPER CYL FWD RS
      OUT     T687 K2  ; NST3_INTERMEDIATE_CYL_FWD_TIMR
; Rung 247
2787  LD      L1396  ; INTERMEDIATE STOPPER CYL BACK RS
      AND     L1397  ; INTERMEDIATE STOPPER CYL FWD RS
      OUT     T688 K20  ; INTERMEDIATE_STOPPER_CYL_LSW_FAI
; Rung 248
2799  LD      T688  ; INTERMEDIATE_STOPPER_CYL_LSW_FAI
      SET     D7075.0  ; NST3_INTERMEDIATE_STOPER_LSW_FAI
; Rung 249
2807  LD      D6000.4  ; NST2_FAULT_RESET
      RST     D7075.0  ; NST3_INTERMEDIATE_STOPER_LSW_FAI
; Rung 250
2815  LD      D7040.0  ; NST3_PRESSING_SLIDE_BACK
      OUT     D7074.0
; Rung 251
2823  LD      D7009.7  ; NST3_EMERG_RET_COMM
      OR      D7079.7
      AND     D5000.0  ; CKT2_AUTO_COTROL
      ANI     D7070.0  ; NST3_INTERMEDIATE_CYL_BACK
      OUT     D7079.7
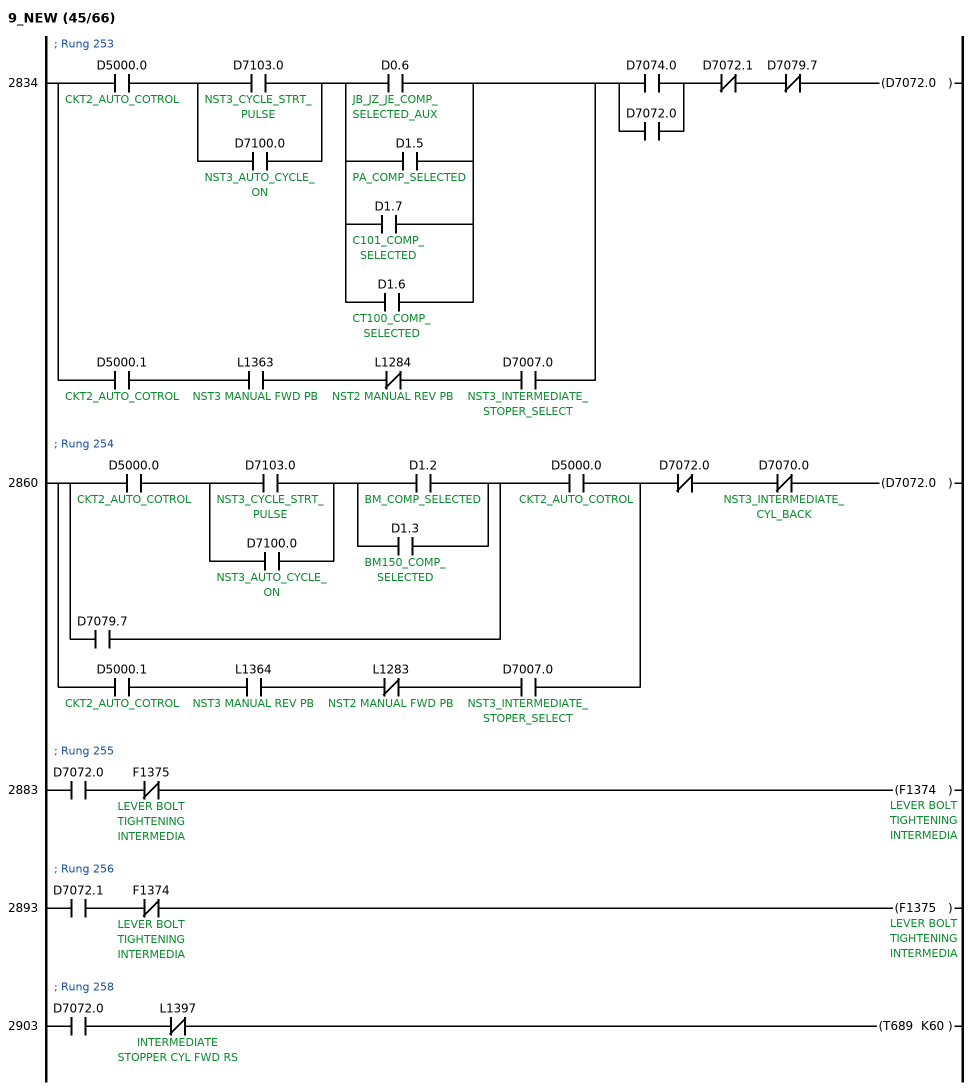
; Rung 253
2834  LD      D5000.0  ; CKT2_AUTO_COTROL
      LD      D7103.0  ; NST3_CYCLE_STRT_PULSE
      OR      D7100.0  ; NST3_AUTO_CYCLE_ON
      ANB
      LD      D0.6  ; JB_JZ_JE_COMP_SELECTED_AUX
      OR      D1.5  ; PA_COMP_SELECTED
      OR      D1.7  ; C101_COMP_SELECTED
      OR      D1.6  ; CT100_COMP_SELECTED
      ANB
      LD      D5000.1  ; CKT2_AUTO_COTROL
      AND     L1363  ; NST3 MANUAL FWD PB
      ANI     L1284  ; NST2 MANUAL REV PB
      AND     D7007.0  ; NST3_INTERMEDIATE_STOPER_SELECT
      ORB
      LD      D7074.0
      OR      D7072.0
      ANB
      ANI     D7072.1
      ANI     D7079.7
      OUT     D7072.0
; Rung 254
2860  LD      D5000.0  ; CKT2_AUTO_COTROL
      LD      D7103.0  ; NST3_CYCLE_STRT_PULSE
      OR      D7100.0  ; NST3_AUTO_CYCLE_ON
      ANB
      LD      D1.2  ; BM_COMP_SELECTED
      OR      D1.3  ; BM150_COMP_SELECTED
      ANB
      OR      D7079.7
      AND     D5000.0  ; CKT2_AUTO_COTROL
      LD      D5000.1  ; CKT2_AUTO_COTROL
      AND     L1364  ; NST3 MANUAL REV PB
      ANI     L1283  ; NST2 MANUAL FWD PB
      AND     D7007.0  ; NST3_INTERMEDIATE_STOPER_SELECT
      ORB
      ANI     D7072.0
      ANI     D7070.0  ; NST3_INTERMEDIATE_CYL_BACK
      OUT     D7072.0
; Rung 255
2883  LD      D7072.0
      ANI     F1375  ; LEVER BOLT TIGHTENING INTERMEDIA
      OUT     F1374  ; LEVER BOLT TIGHTENING INTERMEDIA
; Rung 256
2893  LD      D7072.1
      ANI     F1374  ; LEVER BOLT TIGHTENING INTERMEDIA
      OUT     F1375  ; LEVER BOLT TIGHTENING INTERMEDIA
; Rung 258
2903  LD      D7072.0
      ANI     L1397  ; INTERMEDIATE STOPPER CYL FWD RS
      OUT     T689 K60
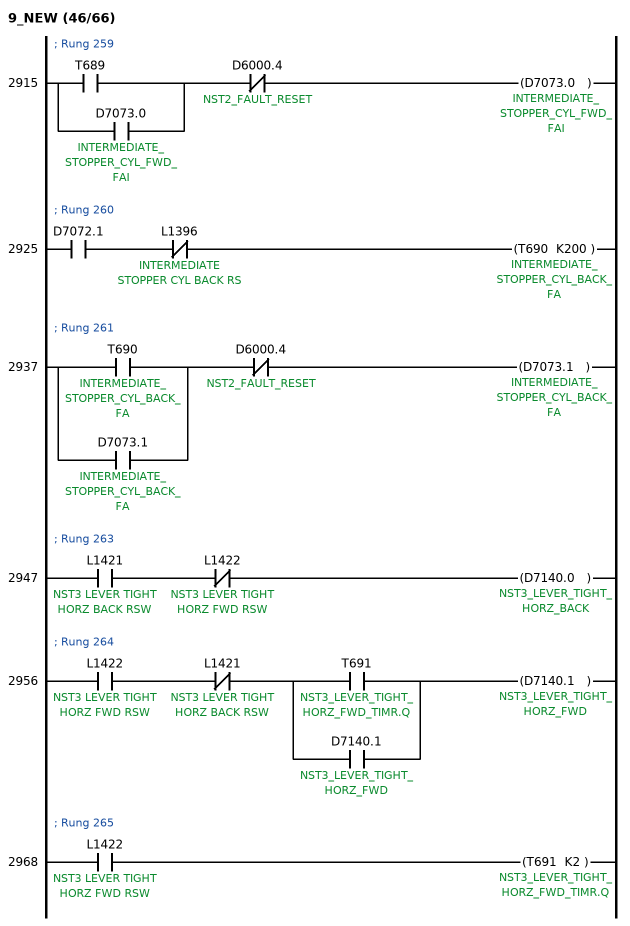
; Rung 259
2915  LD      T689
      OR      D7073.0  ; INTERMEDIATE_STOPPER_CYL_FWD_FAI
      ANI     D6000.4  ; NST2_FAULT_RESET
      OUT     D7073.0  ; INTERMEDIATE_STOPPER_CYL_FWD_FAI
; Rung 260
2925  LD      D7072.1
      ANI     L1396  ; INTERMEDIATE STOPPER CYL BACK RS
      OUT     T690 K200  ; INTERMEDIATE_STOPPER_CYL_BACK_FA
; Rung 261
2937  LD      T690  ; INTERMEDIATE_STOPPER_CYL_BACK_FA
      OR      D7073.1  ; INTERMEDIATE_STOPPER_CYL_BACK_FA
      ANI     D6000.4  ; NST2_FAULT_RESET
      OUT     D7073.1  ; INTERMEDIATE_STOPPER_CYL_BACK_FA
; Rung 263
2947  LD      L1421  ; NST3 LEVER TIGHT HORZ BACK RSW
      ANI     L1422  ; NST3 LEVER TIGHT HORZ FWD RSW
      OUT     D7140.0  ; NST3_LEVER_TIGHT_HORZ_BACK
; Rung 264
2956  LD      L1422  ; NST3 LEVER TIGHT HORZ FWD RSW
      ANI     L1421  ; NST3 LEVER TIGHT HORZ BACK RSW
      LD      T691  ; NST3_LEVER_TIGHT_HORZ_FWD_TIMR.Q
      OR      D7140.1  ; NST3_LEVER_TIGHT_HORZ_FWD
      ANB
      OUT     D7140.1  ; NST3_LEVER_TIGHT_HORZ_FWD
; Rung 265
2968  LD      L1422  ; NST3 LEVER TIGHT HORZ FWD RSW
      OUT     T691 K2  ; NST3_LEVER_TIGHT_HORZ_FWD_TIMR.Q
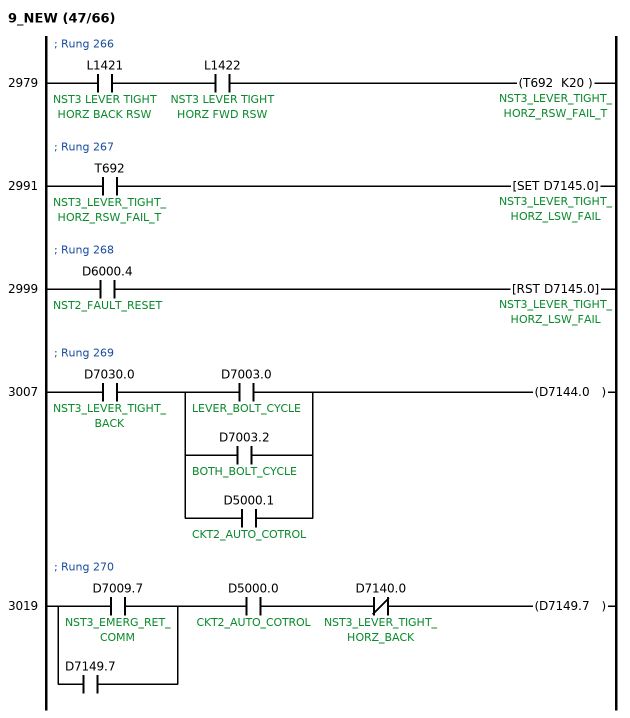
; Rung 266
2979  LD      L1421  ; NST3 LEVER TIGHT HORZ BACK RSW
      AND     L1422  ; NST3 LEVER TIGHT HORZ FWD RSW
      OUT     T692 K20  ; NST3_LEVER_TIGHT_HORZ_RSW_FAIL_T
; Rung 267
2991  LD      T692  ; NST3_LEVER_TIGHT_HORZ_RSW_FAIL_T
      SET     D7145.0  ; NST3_LEVER_TIGHT_HORZ_LSW_FAIL
; Rung 268
2999  LD      D6000.4  ; NST2_FAULT_RESET
      RST     D7145.0  ; NST3_LEVER_TIGHT_HORZ_LSW_FAIL
; Rung 269
3007  LD      D7030.0  ; NST3_LEVER_TIGHT_BACK
      LD      D7003.0  ; LEVER_BOLT_CYCLE
      OR      D7003.2  ; BOTH_BOLT_CYCLE
      OR      D5000.1  ; CKT2_AUTO_COTROL
      ANB
      OUT     D7144.0
; Rung 270
3019  LD      D7009.7  ; NST3_EMERG_RET_COMM
      OR      D7149.7
      AND     D5000.0  ; CKT2_AUTO_COTROL
      ANI     D7140.0  ; NST3_LEVER_TIGHT_HORZ_BACK
      OUT     D7149.7
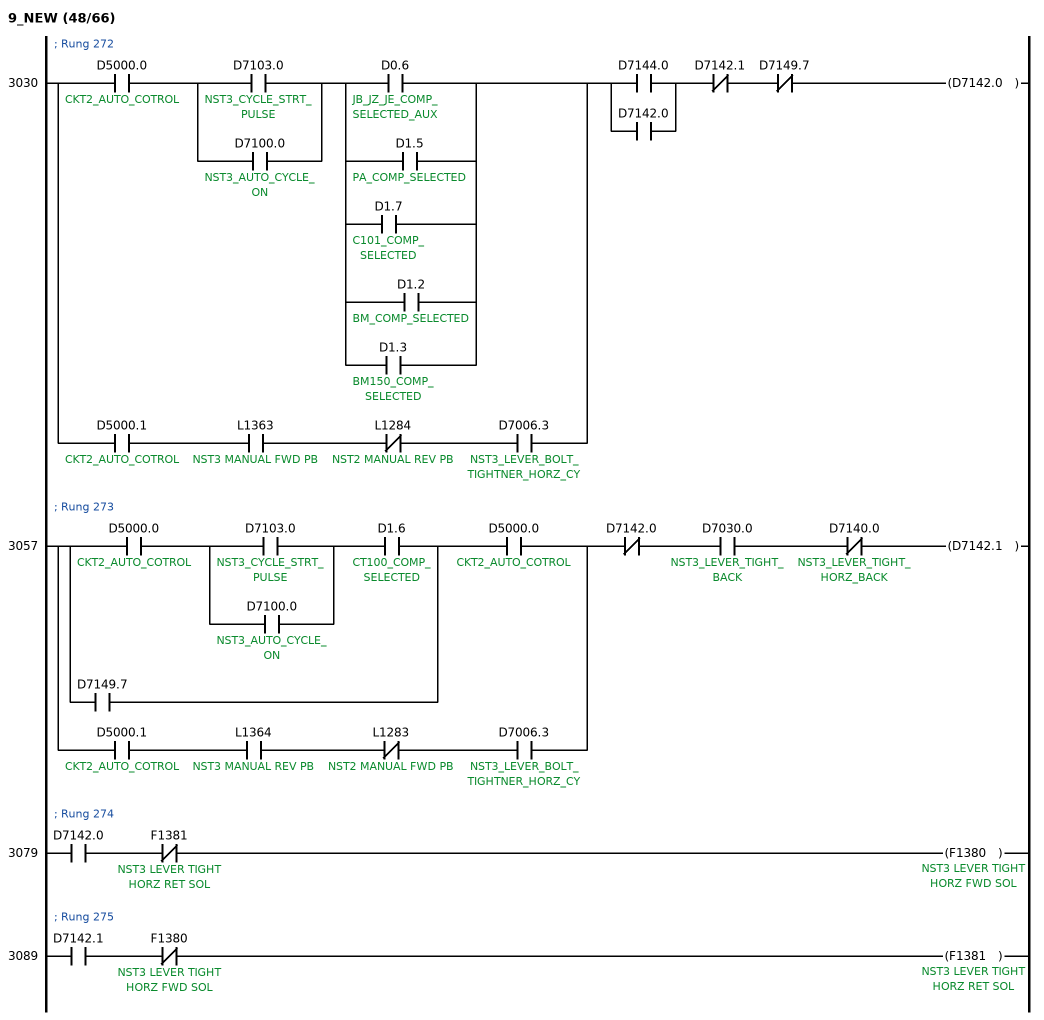
; Rung 272
3030  LD      D5000.0  ; CKT2_AUTO_COTROL
      LD      D7103.0  ; NST3_CYCLE_STRT_PULSE
      OR      D7100.0  ; NST3_AUTO_CYCLE_ON
      ANB
      LD      D0.6  ; JB_JZ_JE_COMP_SELECTED_AUX
      OR      D1.5  ; PA_COMP_SELECTED
      OR      D1.7  ; C101_COMP_SELECTED
      OR      D1.2  ; BM_COMP_SELECTED
      OR      D1.3  ; BM150_COMP_SELECTED
      ANB
      LD      D5000.1  ; CKT2_AUTO_COTROL
      AND     L1363  ; NST3 MANUAL FWD PB
      ANI     L1284  ; NST2 MANUAL REV PB
      AND     D7006.3  ; NST3_LEVER_BOLT_TIGHTNER_HORZ_CY
      ORB
      LD      D7144.0
      OR      D7142.0
      ANB
      ANI     D7142.1
      ANI     D7149.7
      OUT     D7142.0
; Rung 273
3057  LD      D5000.0  ; CKT2_AUTO_COTROL
      LD      D7103.0  ; NST3_CYCLE_STRT_PULSE
      OR      D7100.0  ; NST3_AUTO_CYCLE_ON
      ANB
      AND     D1.6  ; CT100_COMP_SELECTED
      OR      D7149.7
      AND     D5000.0  ; CKT2_AUTO_COTROL
      LD      D5000.1  ; CKT2_AUTO_COTROL
      AND     L1364  ; NST3 MANUAL REV PB
      ANI     L1283  ; NST2 MANUAL FWD PB
      AND     D7006.3  ; NST3_LEVER_BOLT_TIGHTNER_HORZ_CY
      ORB
      ANI     D7142.0
      AND     D7030.0  ; NST3_LEVER_TIGHT_BACK
      ANI     D7140.0  ; NST3_LEVER_TIGHT_HORZ_BACK
      OUT     D7142.1
; Rung 274
3079  LD      D7142.0
      ANI     F1381  ; NST3 LEVER TIGHT HORZ RET SOL
      OUT     F1380  ; NST3 LEVER TIGHT HORZ FWD SOL
; Rung 275
3089  LD      D7142.1
      ANI     F1380  ; NST3 LEVER TIGHT HORZ FWD SOL
      OUT     F1381  ; NST3 LEVER TIGHT HORZ RET SOL
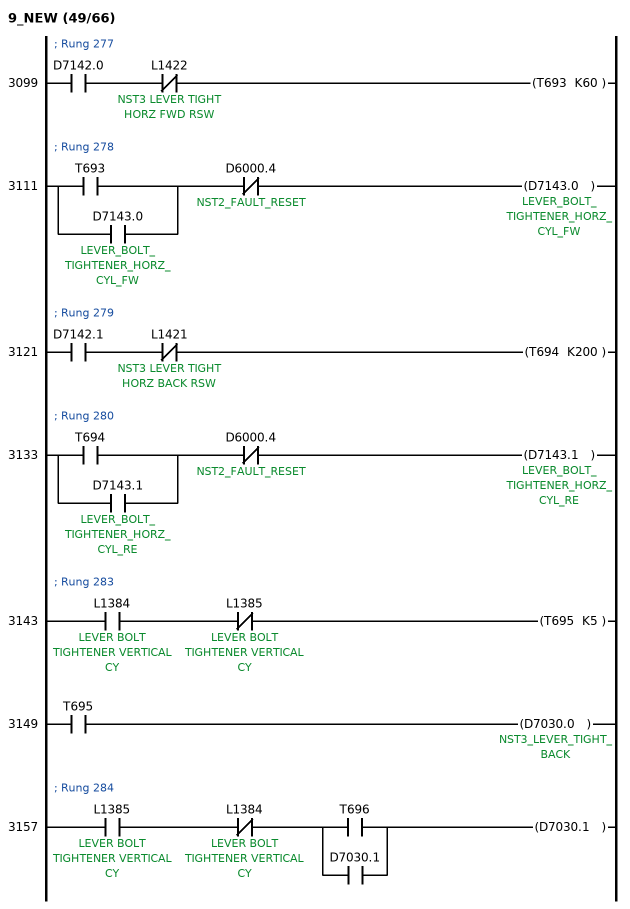
; Rung 277
3099  LD      D7142.0
      ANI     L1422  ; NST3 LEVER TIGHT HORZ FWD RSW
      OUT     T693 K60
; Rung 278
3111  LD      T693
      OR      D7143.0  ; LEVER_BOLT_TIGHTENER_HORZ_CYL_FW
      ANI     D6000.4  ; NST2_FAULT_RESET
      OUT     D7143.0  ; LEVER_BOLT_TIGHTENER_HORZ_CYL_FW
; Rung 279
3121  LD      D7142.1
      ANI     L1421  ; NST3 LEVER TIGHT HORZ BACK RSW
      OUT     T694 K200
; Rung 280
3133  LD      T694
      OR      D7143.1  ; LEVER_BOLT_TIGHTENER_HORZ_CYL_RE
      ANI     D6000.4  ; NST2_FAULT_RESET
      OUT     D7143.1  ; LEVER_BOLT_TIGHTENER_HORZ_CYL_RE
; Rung 283
3143  LD      L1384  ; LEVER BOLT TIGHTENER VERTICAL CY
      ANI     L1385  ; LEVER BOLT TIGHTENER VERTICAL CY
      OUT     T695 K5
3149  LD      T695
      OUT     D7030.0  ; NST3_LEVER_TIGHT_BACK
; Rung 284
3157  LD      L1385  ; LEVER BOLT TIGHTENER VERTICAL CY
      ANI     L1384  ; LEVER BOLT TIGHTENER VERTICAL CY
      LD      T696
      OR      D7030.1
      ANB
      OUT     D7030.1
